{attribute 'GeneratedUsingTerminal: EK1122-0000-0018'}
{attribute addProperty BoxType "EK1122-0000-0018"}
{attribute addProperty Id "Beckhoff_EL32xxsub_EK1100EK1100_1FC0878B2"}
{attribute addProperty CRC "2264526553"}
{attribute addProperty Size "2"}
TYPE Beckhoff_EL32xxEK1122_86F9EED9 EXTENDS EK1122_1FC0878B :
STRUCT
	{attribute addProperty Name "Beckhoff_EL32xxsub_EK1100"}
	{attribute addProperty PreviousPort "Beckhoff EL32xxEK1122 : D"}
	Beckhoff_EL32xxsub_EK1100 : EK1100_1FC0878B;
END_STRUCT
END_TYPE

(* stored: Version 1.2.0.0, ProductVersion 3.1.4024.9
   DUT Beckhoff_EL32xxEK1122_86F9EED9: Id {00cff778-d73f-48aa-9c1a-a015b7bfca33} *)
